// TIA Portal V16 export
// export: Created 2024-05-14T12:25:50.2394744Z, ExportSetting WithDefaults, DisplayName Totally Integrated Automation Portal, DisplayVersion V16, DisplayName TIA Portal Version Control Interface, DisplayVersion V16, DisplayName TIA Portal Openness, DisplayVersion V16, DisplayName STEP 7 Professional, DisplayVersion V16, DisplayName STEP 7 Safety, DisplayVersion V16, DisplayName WinCC Advanced, DisplayVersion V16
DATA_BLOCK "Halcon"   // DB2
{ S7_Optimized_Access := 'TRUE' }
VERSION : 0.1
// stored: AutoNumber true, DBAccessibleFromOPCUA true, IsOnlyStoredInLoadMemory false, IsRetainMemResEnabled false, IsWriteProtectedInAS false, MemoryReserve 100
   VAR
      state : Int;
      "OPC Data" : Struct
         Data_Bool : Bool;
         Data_Integer : Int;
         Data_String : String;
      END_STRUCT;
   END_VAR
BEGIN
END_DATA_BLOCK
